// TIA Portal V17 export
// export: Created 2022-02-03T14:45:13.3263133Z, ExportSetting WithDefaults, DisplayName Totally Integrated Automation Portal, DisplayVersion V17, DisplayName TIA Portal Openness, DisplayVersion V17, DisplayName TIA Portal Version Control Interface, DisplayVersion V17, DisplayName SINAMICS Startdrive Advanced, DisplayVersion V17, DisplayName SINAMICS Startdrive G130, G150, S120, S150, SINAMICS MV, S210, DisplayVersion V17, DisplayName SINAMICS Startdrive G110M, G120, G120C, G120D, G120P, G115D, DisplayVersion V17, DisplayName STEP 7 Professional, DisplayVersion V17, DisplayName STEP 7 Safety, DisplayVersion V17, DisplayName WinCC Advanced, DisplayVersion V17
FUNCTION "StoreStatistics" : Void   // FC6, LAD
VERSION : 0.1
// stored: Access Published, AutoNumber true, IsIECCheckEnabled false, SetENOAutomatically false, UDAEnableTagReadback false
   VAR_INPUT
      new : Bool;
   END_VAR
   VAR_IN_OUT
      store : "typeStore";
      storeStatistics : "typeStoreStatistics";
   END_VAR
   VAR_TEMP
      tempIndex : UInt;
   END_VAR
BEGIN

REGION Network 1
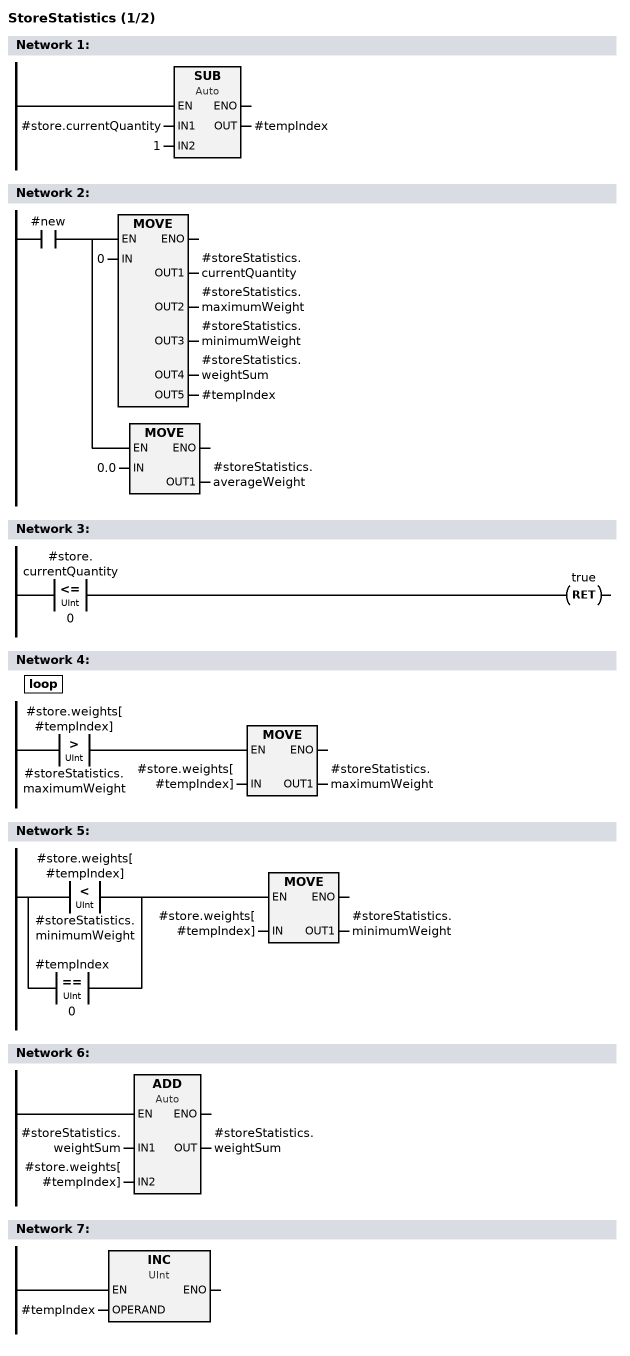
   RUNG wire#powerrail
      Sub(in1 := #store.currentQuantity, in2 := 1, out => #tempIndex)
   END_RUNG
   // the same network as SCL:
   #tempIndex := #store.currentQuantity - 1;
END_REGION

REGION Network 2
   RUNG wire#powerrail
      Contact( #new )
      wire#w1
      Move(in := 0, out1 => #storeStatistics.currentQuantity, out2 => #storeStatistics.maximumWeight, out3 => #storeStatistics.minimumWeight, out4 => #storeStatistics.weightSum, out5 => #tempIndex)
   END_RUNG
   RUNG wire#w1
      Move(in := 0.0, out1 => #storeStatistics.averageWeight)
   END_RUNG
   // the same network as SCL:
   IF #new THEN
       #storeStatistics.currentQuantity := 0;
       #storeStatistics.maximumWeight := 0;
       #storeStatistics.minimumWeight := 0;
       #storeStatistics.weightSum := 0;
       #tempIndex := 0;
       #storeStatistics.averageWeight := 0.0;
   END_IF;
END_REGION

REGION Network 3
   IF #store.currentQuantity <= 0 THEN
       ENO := true;
       RETURN;
   END_IF;
END_REGION

REGION Network 4
   Label( loop )
   RUNG wire#powerrail
      { S7_Templates := "SrcType := UInt" } GT_Contact(in1 := #store.weights[#tempIndex], in2 := #storeStatistics.maximumWeight)
      Move(in := #store.weights[#tempIndex], out1 => #storeStatistics.maximumWeight)
   END_RUNG
   // the same network as SCL:
   loop:
   IF #store.weights[#tempIndex] > #storeStatistics.maximumWeight THEN
       #storeStatistics.maximumWeight := #store.weights[#tempIndex];
   END_IF;
END_REGION

REGION Network 5
   RUNG wire#powerrail
      { S7_Templates := "SrcType := UInt" } LT_Contact(in1 := #store.weights[#tempIndex], in2 := #storeStatistics.minimumWeight)
      wire#w1
      Move(in := #store.weights[#tempIndex], out1 => #storeStatistics.minimumWeight)
   END_RUNG
   RUNG wire#powerrail
      { S7_Templates := "SrcType := UInt" } EQ_Contact(in1 := #tempIndex, in2 := 0)
   END_RUNG wire#w1
   // the same network as SCL:
   IF (#store.weights[#tempIndex] < #storeStatistics.minimumWeight) OR (#tempIndex = 0) THEN
       #storeStatistics.minimumWeight := #store.weights[#tempIndex];
   END_IF;
END_REGION

REGION Network 6
   RUNG wire#powerrail
      Add(in1 := #storeStatistics.weightSum, in2 := #store.weights[#tempIndex], out => #storeStatistics.weightSum)
   END_RUNG
   // the same network as SCL:
   #storeStatistics.weightSum := #storeStatistics.weightSum + #store.weights[#tempIndex];
END_REGION

REGION Network 7
   RUNG wire#powerrail
      { S7_Templates := "DestType := UInt" } Inc( #tempIndex )
   END_RUNG
   // the same network as SCL:
   #tempIndex := #tempIndex + 1;
END_REGION

REGION Network 8
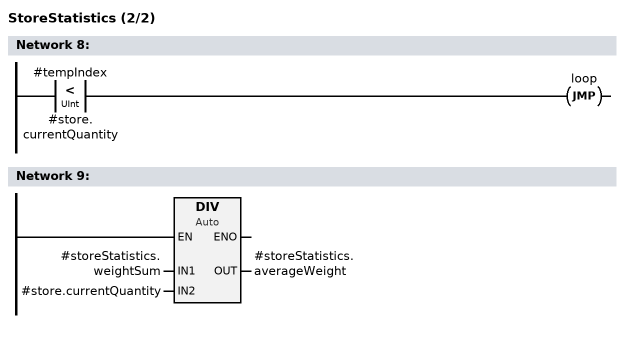
   RUNG wire#powerrail
      { S7_Templates := "SrcType := UInt" } LT_Contact(in1 := #tempIndex, in2 := #store.currentQuantity)
      JumpCoil( loop )
   END_RUNG
   // the same network as SCL:
   IF #tempIndex < #store.currentQuantity THEN GOTO loop; END_IF;
END_REGION

REGION Network 9
   RUNG wire#powerrail
      Div(in1 := #storeStatistics.weightSum, in2 := #store.currentQuantity, out => #storeStatistics.averageWeight)
   END_RUNG
   // the same network as SCL:
   #storeStatistics.averageWeight := #storeStatistics.weightSum / #store.currentQuantity;
END_REGION
END_FUNCTION
